(* PLC project Rasi_feeds_batching.project, Automation Builder 2.7 - Basic Automation Builder 2.7 *)
(* stored: creationDateTime 2026-08-27T18:17:46.8692424, modificationDateTime 2026-08-27T18:17:12.3961725 *)

PROGRAM test_fbd_pou

(* FBD diagram, written out as Structured Text *)
END_PROGRAM
